FUNCTION_BLOCK Resetting_State  IMPLEMENTS ITF_State
VAR_INPUT
END_VAR
VAR_OUTPUT
END_VAR
VAR
	pPML_Base : POINTER TO PML_StatePattern_Base;
	_stateMachine : IPmlStateMachine;
END_VAR

METHOD Cycle : BOOL
VAR_INPUT
END_VAR
_stateMachine.SetStateComplete();
pPML_Base^.SetState(pPML_Base^.idle);
END_METHOD

METHOD FB_init : BOOL
VAR_INPUT
	bInitRetains : BOOL; // if TRUE, the retain variables are initialized (warm start / cold start)
	bInCopyCode : BOOL;  // if TRUE, the instance afterwards gets moved into the copy code (online change)
	pPML_Base : POINTER TO PML_StatePattern_Base;
	statemachine : IPmlStateMachine;
END_VAR
_stateMachine := statemachine;
THIS^.pPML_Base := pPML_Base;
END_METHOD

END_FUNCTION_BLOCK

(* stored: Version 1.1.0.1, ProductVersion 3.1.4024.11
   POU Resetting_State: Id {e487e0e3-f47e-443c-893c-c4527c851321}, SpecialFunc None
   Method Cycle: Id {33253227-e440-4391-8c6c-d0f15e86a992}
   Method FB_init: Id {4facd53f-ccf2-4cc0-b231-e70768116a76} *)
